{attribute 'linkalways'} 
{attribute 'no_explicit_call' := 'This FB is a CLASS and must be accessed using methods or properties'}
{attribute 'enable_dynamic_creation'}
FUNCTION_BLOCK VisionDatatypePack IMPLEMENTS I_DatatypePack
VAR
	// alias
	
	// enums
	_eTcVn2dCodeSearchStrategy : _ETcVn2dCodeSearchStrategy(ETcVn2dCodeSearchStrategy.TCVN_CSS_DEFAULT);
	
	// structures
	_tcVnImageInfo : _TcVnImageInfo;
	_tcVnPixelFormat : _TcVnPixelFormat;
	
	// interface
	_iTcVnImage : _ITcVnImage;
	
END_VAR

METHOD RegisterWith
VAR_INPUT
	Datatypes : I_Datatypes;
END_VAR
// enums
Datatypes.RegisterDatatype(_eTcVn2dCodeSearchStrategy);

// structures
Datatypes.RegisterDatatype(_tcVnImageInfo);
Datatypes.RegisterDatatype(_tcVnPixelFormat);

// interfaces
Datatypes.RegisterDatatype(_iTcVnImage);
END_METHOD

END_FUNCTION_BLOCK

(* stored: Version 1.1.0.1, ProductVersion 3.1.4024.12
   POU VisionDatatypePack: Id {41aa96c4-4e58-0595-14c8-fb1325f46fff}, SpecialFunc None
   Method RegisterWith: Id {5bfb729e-cc5d-077c-086c-02393210cdae} *)
